(* IEC 61131-3 sources: AXOpen/src/components.siemens.identification/app/src, 2 files *)

(* ---- configuration.st ---- *)
USING AXOpen.Components.SIEM.Identification;

CONFIGURATION MyConfiguration
    TASK Main(Interval := T#1ms, Priority := 1);
    PROGRAM P1 WITH Main: MyProgram;

    VAR_GLOBAL
        {S7.extern=ReadWrite}
        sandbox : SandboxContext;
        {S7.extern=ReadWrite}
        documentation : DocumentationContext;
        {S7.extern=ReadWrite}
        _rtc : AXOpen.S71500.Rtc;
    END_VAR
END_CONFIGURATION

(* ---- program.st ---- *)
USING AXOpen.Components.SIEM.Identification;

PROGRAM MyProgram
    VAR_EXTERNAL
        sandbox : SandboxContext;
        documentation : DocumentationContext;
        _rtc : AXOpen.S71500.Rtc;
    END_VAR

    sandbox.Run();
    sandbox.InjectRtc(_rtc);
    documentation.Run();
    documentation.InjectRtc(_rtc);

END_PROGRAM
